{attribute addProperty BoxType "EL2564-0000-0016"}
{attribute addProperty Id "PWM_outputAT %Q*INT162"}
{attribute addProperty CRC "4206222476"}
{attribute addProperty SizeInBites "16"}
{attribute addProperty SizeInBytes "2"}
TYPE PWM_Outputs_Channel_FAB5DC8C :
STRUCT
	{attribute addProperty Name "PWM_output"}
	PWM_output AT %Q* : INT;
END_STRUCT
END_TYPE

(* stored: Version 1.2.0.0, ProductVersion 3.1.4024.9
   DUT PWM_Outputs_Channel_FAB5DC8C: Id {54d0d575-e86c-4c32-9690-e61af6cd11a8} *)
